FUNCTION_BLOCK sT80b
VAR
	_promenlivataNaFilip : BOOL;
	_test : BOOL; 
END_VAR

METHOD  _test
VAR_INPUT
END_VAR
_promenlivataNaFilip:= TRUE;
_test:= FALSE;
END_METHOD

END_FUNCTION_BLOCK

(* stored: Version 1.1.0.1, ProductVersion 3.1.4024.12
   POU sT80b: Id {3cf6e9b3-e801-41fd-874b-1d437fea11c0}, SpecialFunc None
   Method _test: Id {4a5b8f54-185c-4781-84cc-cdd5f85a1e98} *)
